// TIA Portal V20 export
DATA_BLOCK "InstProfinetDeviceDiagStatus"   // DB172
// stored: InstanceOfName LER_DiagnosticsStatus, InstanceOfType FB
"LER_DiagnosticsStatus"
   // VAR_INPUT
   //    devStateHmi_X1 : Array[0..256] of "LAF_typeDevDiagBasic";
   //    devStateHmi_X2 : Array[0..256] of "LAF_typeDevDiagBasic";
   //    UnitSelect : Int;
   //    Reset : Bool;
   // END_VAR
   // VAR_IN_OUT
   //    DevState : "LER_DiagnosticsInterface";
   // END_VAR
   // VAR
   //    staticCntState : Int;
   //    staticCntStartState : Int;
   //    staticCntEndState : Int;
   //    staticCntDev : Int;
   //    staticCntHighLimit_X2 : Array[1..15] of Int;
   //    staticCntLowLimit_X2 : Array[1..15] of Int;
   //    staticCntHighLimit_X1 : Array[1..15] of Int;
   //    staticCntLowLimit_X1 : Array[1..15] of Int;
   //    staticCntModuleState : Int;
   //    staticDevStateError : Array[0..15] of Bool;
   //    statiDevStateMove_X1 : Array[0..15] of Int;
   //    statiDevStateMove_X2 : Array[0..15] of Int;
   // END_VAR
BEGIN
END_DATA_BLOCK
